Staubli VAL3: onEdit.pgx

public program onEdit(string& x_sItem[])
  local num l_nX
  local num l_nY
  local num l_nDelay
begin
  // convert to a num
  toNum(x_sItem,l_nDelay,true)
  // change the field
  call use:insertDialog("Distance [mm] ",l_nDelay,-0.01,2680.01)
  // give back
  if l_nDelay>=0
    l_nDelay=round(l_nDelay)
    x_sItem="AXISMOVEL "+toString("",l_nDelay)
  endIf
end
